(* IEC 61131-3 sources: SCLTeamCoder/experiment/datasets/oscat/oscat_code (part 5) *)

(* ---- STACK_32.st ---- *)
FUNCTION_BLOCK STACK_32
VAR_INPUT
    Din : DWORD;
    E : BOOL := TRUE;
    RD : BOOL;
    WD : BOOL;
    RST : BOOL;
END_VAR

VAR_OUTPUT
    Dout : DWORD;
    EMPTY : BOOL := TRUE;
    FULL : BOOL;
END_VAR

VAR
    stack : ARRAY[0..n] OF DWORD;
    pt : INT;
END_VAR

VAR CONSTANT
    n : INT := 31; // changing this value will change the number of stored elements in the fifo
END_VAR
IF RST THEN
	(* asynchronous reset for the fifo *)
	pt := 0;
	EMPTY := TRUE;
	FULL := FALSE;
	Dout := 0;
ELSIF E THEN
	IF NOT EMPTY AND RD THEN
		(* read one element *)
		pt := pt - 1;
		Dout := stack[pt];
		EMPTY := pt = 0;
		FULL := FALSE;
	END_IF;
	IF NOT FULL AND WD THEN
		(* write one element *)
		stack[pt] := Din;
		pt := pt + 1;
		FULL := pt > n;
		EMPTY := FALSE;
	END_IF;
END_IF;

(* revision history
hm	4. aug. 2006	rev 1.0
	original version

hm	19. feb 2008	rev 1.1
	performance improvements

hm	17. oct. 2008	rev 1.2
	deleted unnecessary init with 0

ks	27. oct. 2008	rev 1.3
	optimized performance

hm	25. jul 2009	rev 2.0
	changed inputs to allow simultsaneous read and write

*)
END_FUNCTION_BLOCK

(* ---- STAIR2.st ---- *)
FUNCTION_BLOCK STAIR2
VAR_INPUT
    X : REAL;
    D : REAL;
END_VAR

VAR_OUTPUT
    Y : REAL;
END_VAR
IF D > 0.0 THEN
	IF X >= Y + D OR X <= Y - D THEN Y := FLOOR(X/D) * D; END_IF;
ELSE
	Y := X;
END_IF;

(* revision history
hm	28 jan 2007		rev 1.0
	original version

hm	27. dec 2007	rev 1.1
	changed code for better performance

hm	30. jun. 2008	rev 1.2
	added type conversions to avoid warnings under codesys 3.0

ks	26. oct. 2008	rev 1.3
	improved code

hm	10. mar. 2009	rev 1.4
	real constants updated to new systax using dot

*)
END_FUNCTION_BLOCK

(* ---- STORE_8.st ---- *)
FUNCTION_BLOCK STORE_8
VAR_INPUT
    Set : BOOL;
    D0 : BOOL;
    D1 : BOOL;
    D2 : BOOL;
    D3 : BOOL;
    D4 : BOOL;
    D5 : BOOL;
    D6 : BOOL;
    D7 : BOOL;
    Clr : BOOL;
    Rst : BOOL;
END_VAR

VAR_OUTPUT
    Q0 : BOOL;
    Q1 : BOOL;
    Q2 : BOOL;
    Q3 : BOOL;
    Q4 : BOOL;
    Q5 : BOOL;
    Q6 : BOOL;
    Q7 : BOOL;
END_VAR

VAR
    edge : BOOL;
END_VAR
IF rst OR set THEN
	q0 := NOT rst;
	q1 := q0;
	q2 := q0;
	q3 := q0;
	q4 := q0;
	q5 := q0;
	q6 := q0;
	q7 := q0;
ELSE
	IF D0 THEN Q0 := TRUE; END_IF;
	IF D1 THEN Q1 := TRUE; END_IF;
	IF D2 THEN Q2 := TRUE; END_IF;
	IF D3 THEN Q3 := TRUE; END_IF;
	IF D4 THEN Q4 := TRUE; END_IF;
	IF D5 THEN Q5 := TRUE; END_IF;
	IF D6 THEN Q6 := TRUE; END_IF;
	IF D7 THEN Q7 := TRUE; END_IF;

	IF clr AND NOT edge THEN
		IF q0 THEN q0 := FALSE;
		ELSIF q1 THEN q1 := FALSE;
		ELSIF q2 THEN q2 := FALSE;
		ELSIF q3 THEN q3 := FALSE;
		ELSIF q4 THEN q4 := FALSE;
		ELSIF q5 THEN q5 := FALSE;
		ELSIF q6 THEN q6 := FALSE;
		ELSE q7 := FALSE;
		END_IF;
	END_IF;
	edge := clr;
END_IF;

(* revision history
hm	25.12.2007	rev 1.0
	original version

hm	30. oct. 2008	rev 1.1
	optimized performance

hm	14. mar. 2009	rev 1.2
	removed double assignments

*)
END_FUNCTION_BLOCK

(* ---- SUN_POS.st ---- *)
FUNCTION_BLOCK SUN_POS
VAR_INPUT
    latitude : REAL;  // latitude of geographical position
    longitude : REAL; // longitude of geographical position
    utc : DT;        // world time
END_VAR

VAR_OUTPUT
    B : REAL;
    H : REAL;
    HR : REAL;
END_VAR

VAR
    g : REAL;
    a : REAL;
    d : REAL;
    t1 : REAL;
    n : REAL;
    e : REAL;
    c : REAL;
    tau : REAL;
    sin_d : REAL;
    rlat : REAL;
    sin_lat : REAL;
    cos_lat : REAL;
    cos_tau : REAL;
    cos_d : REAL;
END_VAR
(* n is the julian date and the number of days since 1.1.2000-12:00 midday *)
(* be careful for step7 date startes 1.1.1990 instead of 1.1.1970 *)
(* for step7 this line must change *)
n := DWORD_TO_REAL(DT_TO_DWORD(UTC) - 946728000) * 0.000011574074074074;
g :=MODR(6.240040768 + 0.01720197 * n, math.PI2);
d := MODR(4.89495042 + 0.017202792 * n, math.PI2) + 0.033423055 * SIN(g) + 0.000349066 * SIN(2.0*g);
e := 0.409087723 - 0.000000006981317008 * n;
cos_d := COS(d);
sin_d := SIN(d);
a := ATAN(COS(e) * sin_d / cos_d);
IF cos_d < 0.0 THEN a := a + math.PI; END_IF;
c := ASIN(SIN(e) * sin_d);

(* also here we must be very careful utc is from 1.1.1970 for step7 the formula must change *)
tau := RAD(MODR(6.697376 + (n - 0.25) * 0.0657098245037645 + DWORD_TO_REAL(TOD_TO_DWORD(DT_TO_TOD(utc))) * 0.0000002785383333, 24.0) * 15.0 + longitude) - a;
rlat := RAD(latitude);
sin_lat := SIN(rlat);
cos_lat := COS(rlat);
cos_tau := COS(tau);
t1 := cos_tau * sin_lat - TAN(c) * cos_lat;
B := ATAN(SIN(tau) / t1);
IF t1< 0.0 THEN B := B + math.PI2; ELSE B := B + math.PI; END_IF;
B := DEG(MODR(B, math.PI2));
h := DEG(ASIN(COS(C) * cos_tau * cos_lat +SIN(c) * sin_lat));
IF h > 180.0 THEN h := h - 360.0; END_IF;
(* consider refraction *)
HR := h + REFRACTION(h);

(* revision history
hm	1. feb 2007	rev 1.0
	original version

hm	6. jan 2008	rev 1.1
	performance improvements

hm	18. jan 2008	rev 1.2
	further performance improvements
	only calculate once every 10 seconds

hm	16. mar. 2008	rev 1.3
	added type conversion to avoid warnings under codesys 3.0

hm	30. jun. 2008	rev 1.4
	added type conversions to avoid warnings under codesys 3.0

hm	18. oct. 2008	rev 1.5
	using math constants

hm	17. dec. 2008	rev 1.6
	angles below horizon are displayed in negative degrees

hm	27. feb. 2009	rev 2.0
	new code with better accuracy

hm	7. mar. 2009	rev 2.1
	refraction is added after angle normalization
	deleted 10 second lockout
	added output for astronomical heigth h
*)
END_FUNCTION_BLOCK

(* ---- SUN_TIME.st ---- *)
FUNCTION_BLOCK SUN_TIME
// Input Variables
VAR_INPUT
    LATITUDE : REAL; // latitude of geographical position
    LONGITUDE : REAL; // longitude of geographical position
    UTC : DATE; // world time
    H : REAL := -0.83333333333; // heighth above horizon for sunrise
END_VAR

// Output Variables
VAR_OUTPUT
    MIDDAY : TOD; // astrological midday in hours when sun stands at south direction
    SUN_RISE : TOD; // sun rise for current day in local time
    SUN_SET : TOD; // sun set for current day in local time
    SUN_DECLINATION : REAL; // sun declination above horizon at midday in degrees
END_VAR

// Local Variables
VAR
    dk : REAL; // sun declination at midday
    delta : TIME; // delta from midday for sunrise and sunset
    b : REAL;
END_VAR
B := latitude * 0.0174532925199433;
MIDDAY := SUN_MIDDAY(longitude, utc);
DK := 0.40954 * SIN(0.0172 * (INT_TO_REAL(DAY_OF_YEAR(utc)) - 79.35));
sun_declination := DEG(DK);
IF sun_declination > 180.0 THEN sun_declination := sun_declination - 360.0; END_IF;
sun_declination := 90.0 - LATITUDE + sun_declination;
delta := HOUR_TO_TIME(ACOS((SIN(RAD(H)) - SIN(B) * SIN(DK)) / (COS(B) * COS(DK))) * 3.819718632);
sun_rise := MIDDAY - delta;
sun_set := MIDDAY + delta;

(* revision history

rev 1.1	hm	20.1.2007
	deleted unused variables sun_riseR and sun_setR

rev 1.2 hm 17.4.2007
	corrected error while sun:midday would not be corrected for longitude.

rev 1.3	hm	6. jan 2008
	performance improvements

rev	1.4 hm	17. jan 2008
	calculation is now only performed once a day

hm	10. mar. 2009	rev 1.5
	improved performance
	calculation will be performed on every call to allow movong installations

hm	26. jul 2009	rev 1.6
	fixed a problem with wrong midday calculation

hm	25. jan. 2011	rev 1.7
	using function sun_midday
	corrected angle of sun_declination
	added input H
*)
END_FUNCTION_BLOCK

(* ---- TC_MS.st ---- *)
FUNCTION_BLOCK TC_MS
VAR_OUTPUT
    TC : DWORD;
END_VAR

VAR
    init : BOOL;
    tx : DWORD;
    last : DWORD;
END_VAR
(* read system timer *)
tx := T_PLC_MS();

IF NOT init THEN
	init := TRUE;
	TC := 0;
ELSE
	tc := tx - last;
END_IF;
last := tx;

(* revision history
hm		13. mar. 2008	rev 1.0
	original version

*)
END_FUNCTION_BLOCK

(* ---- TC_S.st ---- *)
FUNCTION_BLOCK TC_S
VAR_OUTPUT
    TC : REAL;
END_VAR

VAR
    init : BOOL;
    tx : DWORD;
    last : DWORD;
END_VAR
(* read system timer *)
tx := T_PLC_US();

IF NOT init THEN
	init := TRUE;
	TC := 0.0;
ELSE
	tc := DWORD_TO_REAL(tx - last)*1.0E-6;
END_IF;
last := tx;

(* revision history
hm	13. mar. 2008	rev 1.0
	original version

hm	16. mar 2008	rev 1.1
	added type conversion to avoid warnings under codesys 3.0

hm	11. mar. 2009	rev 1.2
	changed real constants to use dot syntax

*)
END_FUNCTION_BLOCK

(* ---- TC_US.st ---- *)
FUNCTION_BLOCK TC_US
VAR_OUTPUT
    TC : DWORD;
END_VAR

VAR
    init : BOOL;
    tx : DWORD;
    last : DWORD;
END_VAR
(* read system timer *)
tx := T_PLC_US();

IF NOT init THEN
	init := TRUE;
	TC := 0;
ELSE
	tc := tx - last;
END_IF;
last := tx;

(* revision history
hm		13. mar. 2008	rev 1.0
	original version

*)
END_FUNCTION_BLOCK

(* ---- TEMPERATURE.st ---- *)
FUNCTION_BLOCK TEMPERATURE
VAR_INPUT
    K : REAL;
    C : REAL := -273.15;
    F : REAL := -459.67;
    Re : REAL := -218.52;
    Ra : REAL;
END_VAR

VAR_OUTPUT
    YK : REAL;
    YC : REAL;
    YF : REAL;
    YRe : REAL;
    YRa : REAL;
END_VAR
YK := K + (C + 273.15) + (F + 459.67) * 0.555555555555 + (Re * 1.25 + 273.15) + (Ra * 0.555555555555);
YC := YK -273.15;
YF := YK * 1.8 - 459.67;
YRe := (YK - 273.15) * 0.8;
YRa := YK * 1.8;

(* revision history
hm	21. feb. 2008	rev 1.0
	original version

*)
END_FUNCTION_BLOCK

(* ---- TICKER.st ---- *)
FUNCTION_BLOCK TICKER
VAR_INPUT
    N : INT;
    PT : TIME;
END_VAR

VAR_IN_OUT
    Text : STRING[STRING_LENGTH];
END_VAR

VAR_OUTPUT
    Display : STRING[STRING_LENGTH];
END_VAR

VAR
    delay : TP;
    step : INT;
END_VAR
(* generate next ticker when delay is low *)
IF N < LEN(text) THEN
	IF NOT delay.Q THEN
		(* increase step for next tick *)
		step := step + 1;
		IF step > LEN(text) THEN step := 1; END_IF;
		(* extract dispay from text *)
		display := MID(text, N, step);
		(* set delay timer for next tick *)
		delay(in := TRUE, PT := PT);
	ELSE;
		(* execute delay timer *)
		delay(in := FALSE);
	END_IF;
ELSE
	display := text;
END_IF;
(* revision history
hm	4. dec. 2007	rev 1.0
	original version

hm	15. dec. 2007	rev 1.1
	step now starts at 1 instaed of 0

hm	29. mar. 2008	rev 1.2
	changed STRING to STRING(STRING_LENGTH)
*)
END_FUNCTION_BLOCK

(* ---- TMAX.st ---- *)
FUNCTION_BLOCK TMAX
VAR_INPUT
    IN     : BOOL;
    PT     : TIME;
END_VAR

VAR_OUTPUT
    Q      : BOOL;
    Z      : BOOL;
END_VAR

VAR
    tx      : TIME;
    start    : TIME;
    last_in  : BOOL;
END_VAR
(* read system timer *)
tx := DWORD_TO_TIME(T_PLC_MS());

Z := FALSE;

IF NOT in THEN
	Q := FALSE;
ELSIF IN AND NOT last_in THEN
	Q := TRUE;
	start := tx;
ELSIF (tx - start >= PT) AND Q THEN
	Q := FALSE;
	Z := TRUE;
END_IF;

last_in := IN;

(* revision history
hm	20. jul. 2008	rev 1.0
	original version

*)
END_FUNCTION_BLOCK

(* ---- TMIN.st ---- *)
FUNCTION_BLOCK TMIN
VAR_INPUT
    IN : BOOL;
    PT : TIME;
END_VAR

VAR_OUTPUT
    Q : BOOL;
END_VAR

VAR
    pm : TP;  // Assuming TP is a previously defined derived type
END_VAR
pm(in := IN, PT := PT);
Q := IN OR pm.Q;

(* revision history
hm	21. jul. 2008	rev 1.0
	original version

*)
END_FUNCTION_BLOCK

(* ---- TOF_1.st ---- *)
FUNCTION_BLOCK TOF_1
VAR_INPUT
    IN : BOOL;
    PT : TIME;
    RST : BOOL;
END_VAR

VAR_OUTPUT
    Q : BOOL;
END_VAR

VAR
    tx : TIME;
    start : TIME;
END_VAR
(* read system timer *)
tx := DWORD_TO_TIME(T_PLC_MS());

IF RST THEN
	Q := FALSE;
ELSIF IN THEN
	Q := TRUE;
	start := tx;
ELSIF tx - start >= PT THEN
	Q := FALSE;
END_IF;

(* revision history
hm	17. jul. 2008	rev 1.0
	original version

*)
END_FUNCTION_BLOCK

(* ---- TOGGLE.st ---- *)
FUNCTION_BLOCK TOGGLE
VAR_INPUT
    CLK : BOOL;
    rst : BOOL;
END_VAR

VAR_OUTPUT
    Q : BOOL;
END_VAR

VAR
    edge : BOOL;
END_VAR
IF rst THEN
	q := 0;
ELSIF clk AND NOT edge THEN
	Q := NOT Q;
END_IF;
edge := clk;

(* revision history

hm	13.9.2007		rev 1.0
	original version

hm	30. oct. 2008	rev 1.1
	deleted unnecessary init

*)
END_FUNCTION_BLOCK

(* ---- TONOF.st ---- *)
FUNCTION_BLOCK TONOF
VAR_INPUT
    IN : BOOL;
    T_ON : TIME;
    T_OFF : TIME;
END_VAR

VAR_OUTPUT
    Q : BOOL;
END_VAR

VAR
    X : TON; // Assuming TON is a defined timer structure in your environment
    old : BOOL;
    mode : BOOL;
END_VAR
IF IN XOR old THEN
  X(IN := FALSE, PT := SEL(IN,T_OFF,T_ON));
  mode := IN;
  old := IN;
END_IF;
X(IN := TRUE);
IF X.Q THEN Q := mode;END_IF;

(* revision history
hm	10. dec 2007	rev 1.0
	original version

hm	17. sep. 2007	rev 1.1
	improved performance

hm	21. jul. 2009	rev 1.2
	fixed a timing probelm

*)
END_FUNCTION_BLOCK

(* ---- TP_1.st ---- *)
FUNCTION_BLOCK TP_1
VAR_INPUT
    IN : BOOL;
    PT : TIME;
    RST : BOOL;
END_VAR

VAR_OUTPUT
    Q : BOOL;
END_VAR

VAR
    tx : TIME;
    start : TIME;
    ix : BOOL;
END_VAR
(* read system timer *)
tx := DWORD_TO_TIME(T_PLC_MS());

IF RST THEN
	Q := FALSE;
ELSIF IN AND NOT ix THEN
	Q := TRUE;
	start := tx;
ELSIF tx - start >= PT THEN
	Q := FALSE;
END_IF;

ix:= IN;

(* revision history
hm	28. jun. 2008
	original version

*)
END_FUNCTION_BLOCK

(* ---- TP_1D.st ---- *)
FUNCTION_BLOCK TP_1D
VAR_INPUT
    IN : BOOL;
    PT1 : TIME;
    PTD : TIME;
    RST : BOOL;
END_VAR

VAR_OUTPUT
    Q : BOOL;
    W : BOOL;
END_VAR

VAR
    tx : TIME;
    start : TIME;
    ix : BOOL;
END_VAR
(* read system timer *)
tx := DWORD_TO_TIME(T_PLC_MS());

IF RST THEN
	Q := FALSE;
	rst := FALSE;
	W := FALSE;
ELSIF W THEN
	IF tx - start >= PTD THEN
		W := FALSE;
	END_IF;
ELSIF IN AND NOT ix THEN
	Q := TRUE;
	start := tx;
	in := FALSE;
ELSIF tx - start >= PT1 THEN
	Q := FALSE;
	W := TRUE;
	start := tx;
END_IF;

ix := IN;

(* revision history
hm	28. jun. 2008
	original version

*)
END_FUNCTION_BLOCK

(* ---- TP_X.st ---- *)
FUNCTION_BLOCK TP_X
VAR_INPUT
    IN : BOOL;
    PT : TIME;
END_VAR

VAR_OUTPUT
    Q : BOOL;
    ET : TIME;
END_VAR

VAR
    edge : BOOL;
    start : TIME;
    tx : TIME;
END_VAR
(* read system_time *)
tx := DWORD_TO_TIME(T_PLC_MS());

(* rising edge trigger *)
IF IN AND NOT edge THEN
	start := tx;
	Q := PT > t#0ms;
ELSIF Q THEN
	ET := tx - start;
	IF ET >= PT THEN
		Q := FALSE;
		ET := t#0ms;
	END_IF;
END_IF;
edge := IN;

(* revision history
hm	4. aug 2006		rev 1.0
	original version

hm	17. sep 2007	rev 1.1
	replaced time() with T_PLC_MS() for compatibility reasons

hm	19. oct. 2008	rev 1.2
	renamed to TP_R to TP_X for compatibility reasons

hm	17. dec. 2008	rev 1.3
	code optimized

*)
END_FUNCTION_BLOCK

(* ---- TREND.st ---- *)
FUNCTION_BLOCK TREND
VAR_INPUT
    X : REAL;  // Input variable
END_VAR

VAR_OUTPUT
    Q : BOOL;  // Output variable
    TU : BOOL; // Output variable
    TD : BOOL; // Output variable
    D : REAL;  // Output variable
END_VAR

VAR
    last_X : REAL;  // Local variable
END_VAR
TU := X > last_X;
TD := X < last_X;
Q := TU OR TD;
D := X - LAST_X;

last_X := X;

(* revision history
hm	21. aug. 2009	rev 1.0
	original version

*)
END_FUNCTION_BLOCK

(* ---- TREND_DW.st ---- *)
FUNCTION_BLOCK TREND_DW
VAR_INPUT
    X : DWORD;
END_VAR
VAR_OUTPUT
    Q : BOOL;
    TU : BOOL;
    TD : BOOL;
    D : DWORD;
END_VAR
VAR
    last_X : DWORD;
END_VAR
IF X > last_X THEN
	TU := TRUE;
	TD := FALSE;
	D := X - last_X;
	Q := TRUE;
ELSIF X < last_X THEN
	TD := TRUE;
	TU := FALSE;
	D := last_X - X;
	Q := FALSE;
ELSE
	TU := FALSE;
	TD := FALSE;
	D := 0;
END_IF;
last_X := X;

(* revision history
hm	21. nov. 2008	rev 1.0
	original version

hm	20. feb. 2009	rev 1.1
	added outputs TU, TD and D

hm	14. mar. 2009	rev 1.2
	removed double assignments

*)
END_FUNCTION_BLOCK

(* ---- TUNE.st ---- *)
FUNCTION_BLOCK TUNE
VAR_INPUT
    SET : BOOL;
    SU : BOOL;
    SD : BOOL;
    RST : BOOL;
    SS : REAL := 0.1;
    Limit_L : REAL;
    LIMIT_H : REAL := 100.0;
    RST_val : REAL;
    SET_val : REAL := 100.0;
    T1 : TIME := TIME#500ms;
    T2 : TIME := TIME#2s0ms;
    S1 : REAL := 2.0;
    S2 : REAL := 10.0;
END_VAR_INPUT

VAR_OUTPUT
    Y : REAL;
END_VAR_OUTPUT

VAR
    tx : DWORD;
    start : DWORD;
    start2 : DWORD;
    state : INT;
    in : BOOL;
    step : REAL;
    SPEED : REAL;
    Y_start : REAL;
    Y_start2 : REAL;
END_VAR
(* read system time *)
tx := T_PLC_MS();

IF rst THEN
	Y := RST_val;
	state := 0;
ELSIF set THEN
	Y := SET_val;
	state := 0;
ELSIF state > 0 THEN
	(* key has been pushed state machine operating *)
	(* first read the correct input *)
	IF state = 1 THEN
		(* step up *)
		in := su;
	ELSE
		(* step down *)
		in := sd;
	END_IF;
	(* check for single step operation *)
	IF NOT in AND tx - start <= TIME_TO_DWORD(T1) THEN
		Y := Y_start + step;
		state := 0;
	(* check if fast ramp needs to be generated *)
	ELSIF in AND tx - start >= TIME_TO_DWORD(T2) THEN
		Y := Y_start2 + DWORD_TO_REAL(tx - start2) * s2 / speed;
	(* check if slow ramp needs to be generated *)
	ELSIF in AND tx - start >= TIME_TO_DWORD(T1) THEN
		Y := Y_start + DWORD_TO_REAL(tx - start - TIME_TO_DWORD(T1)) * S1 / speed;
		start2 := tx;
		Y_start2 := Y;
	ELSIF NOT in THEN
		state := 0;
	END_IF;
ELSIF su THEN
	(* slow step up *)
	state := 1;
	start := tx;
	step := ss;
	speed := 1000.0;
	Y_start := Y;
ELSIF sd THEN
	(* slow step down *)
	state := 2;
	start := tx;
	step := -ss;
	speed := -1000.0;
	Y_start := Y;
END_IF;

(* make sure output does not exceed limits *)
Y := LIMIT(LIMIT_L, Y, LIMIT_H);

(* revision history
hm	3.11.2007		rev 1.0
	original version

hm	16. mar. 2008	rev 1.1
	added type conversions to avoid warnings under codesys 3.0

hm	11. mar. 2009	rev 1.2
	real constants updated to new systax using dot

*)
END_FUNCTION_BLOCK

(* ---- TUNE2.st ---- *)
FUNCTION_BLOCK TUNE2
VAR_INPUT
    SET     : BOOL;
    SU      : BOOL;
    SD      : BOOL;
    FU      : BOOL;
    FD      : BOOL;
    RST     : BOOL;
    SS      : REAL := 0.1;
    FS      : REAL := 5.0;
    Limit_L : REAL;
    LIMIT_H : REAL := 100.0;
    RST_val : REAL;
    SET_val : REAL := 100.0;
    TR      : TIME := TIME#500ms;
    S1      : REAL := 2.0;
    S2      : REAL := 10.0;
END_VAR

VAR_OUTPUT
    Y       : REAL;
END_VAR

VAR
    tx      : DWORD;
    start    : DWORD;
    state   : INT;
    in      : BOOL;
    step    : REAL;
    SPEED   : REAL;
    Y_start : REAL;
END_VAR
(* read system time *)
tx := T_PLC_MS();

IF rst THEN
	Y := RST_val;
	state := 0;
ELSIF set THEN
	Y := SET_val;
	state := 0;
ELSIF state > 0 THEN
	(* key has been pushed state machine operating *)
	(* first read the correct input *)
	CASE state OF
		1 :	(* slow up *)
			in := su;
		2 :	(* slow down *)
			in := sd;
		3 :	(* fast up *)
			in := fu;
		4 :	(* fast down *)
			in := fd;
	END_CASE;
	(* check for single step operation *)
	IF NOT in AND tx - start <= TIME_TO_DWORD(TR) THEN
		Y := Y_start + step;
		state := 0;
	(* check if ramp needs to be generated *)
	ELSIF in AND tx - start >= TIME_TO_DWORD(TR) THEN
		Y := Y_start + DWORD_TO_REAL(tx - start - TIME_TO_DWORD(TR)) * speed;
	ELSIF NOT in THEN
		state := 0;
	END_IF;
ELSIF su THEN
	(* slow step up *)
	state := 1;
	start := tx;
	step := ss;
	speed := s1 * 1.0E-3;
	Y_start := Y;
ELSIF sd THEN
	(* slow step down *)
	state := 2;
	start := tx;
	step := -ss;
	speed := -s1 * 1.0E-3;
	Y_start := Y;
ELSIF fu THEN
	(* fast step up *)
	state := 3;
	start := tx;
	step := fs;
	speed := s2 * 1.0E-3;
	y_start := Y;
ELSIF fd THEN
	(* fast step down *)
	state := 4;
	start := tx;
	step := -fs;
	speed := -s2 * 1.0E-3;
	y_start := Y;
END_IF;

(* make sure output does not exceed limits *)
Y := LIMIT(LIMIT_L, Y, LIMIT_H);

(* revision history
hm	3.11.2007		rev 1.0
	original version

hm	16. 3. 2008	rev 1.1
	added type conversions to avoid warnings in codesys 3.0
	improved performance

hm	11. mar. 2009	rev 1.2
	real constants updated to new systax using dot

*)
END_FUNCTION_BLOCK
